Fanuc KAREL source: CLR_PORT_SIM.kl

PROGRAM T
%NOLOCKGROUP
VAR
 v0 : INTEGER
 v1 : INTEGER
 v2 : INTEGER
BEGIN
 CLR_PORT_SIM(v0, v1, v2)
END T
